(* PLC project Garden Watering, CODESYS CODESYS V3.5 SP14 Patch 1, author Toni Kucic *)
(* stored: creationDateTime 2019-07-15T20:33:55.3489661, version 1.0, modificationDateTime 2019-07-15T20:33:55.2060528, organization TK Automation *)

PROGRAM xc02_GardenWatering
  VAR
    vFlowersXY : ARRAY[0..59, 0..1] OF INT := [276, 253, 381, 253, 486, 253, 591, 253, 696, 253, 801, 253, 906, 253, 1011, 253, 1116, 253, 1221, 253, 276, 354, 381, 354, 486, 354, 591, 354, 696, 354, 801, 354, 906, 354, 1011, 354, 1116, 354, 1221, 354, 276, 455, 381, 455, 486, 455, 591, 455, 696, 455, 801, 455, 906, 455, 1011, 455, 1116, 455, 1221, 455, 276, 556, 381, 556, 486, 556, 591, 556, 696, 556, 801, 556, 906, 556, 1011, 556, 1116, 556, 1221, 556, 276, 667, 381, 667, 486, 667, 591, 667, 696, 667, 801, 667, 906, 667, 1011, 667, 1116, 667, 1221, 667, 276, 768, 381, 768, 486, 768, 591, 768, 696, 768, 801, 768, 906, 768, 1011, 768, 1116, 768, 1221, 768];
    vManual : BOOL;  (* Coordinates of flowers in format Flower0 -x,y *)
    vXCMD : REAL;
    vYCMD : REAL;
    i : INT;
    Watering : TON;
    ActuatorOverFlower : CollisionDetection;
  END_VAR

                    (* Control from the graphics *)
IF NOT xgv02.Remote THEN
	xgv02.HorizontalLeft := xgv02.HMIDownLeft OR xgv02.HMILeft OR xgv02.HMIUpLeft;
	xgv02.HorizontalRight := xgv02.HMIDownRight OR xgv02.HMIRight OR xgv02.HMIUpRight;
	xgv02.VerticalUp := xgv02.HMIUpLeft OR xgv02.HMIUp OR xgv02.HMIUpRight;
	xgv02.VerticalDown := xgv02.HMIDownLeft OR xgv02.HMIDown OR xgv02.HMIDownRight;
	xgv02.OpenWaterValve := xgv02.HMIOpenWater;
END_IF;

(* Coordinate control *)
IF xgv02.Remote AND vManual THEN
	vXCMD := xgv02.HMICoorXCmd;
	vYCMD := xgv02.HMICoorYCmd;
ELSE
	xgv02.HMICoorXCmd := xgv02.PositionX;
	xgv02.HMICoorYCmd := xgv02.PositionY;
END_IF

(* Full automatic algorithm *)
IF xgv02.Remote AND NOT vManual THEN
	vXCMD := vFlowersXY[i,0]+ 30;
	vYCMD := vFlowersXY[i,1]+ 30;
	
	ActuatorOverFlower(
		xcor1:= xgv02.PositionX, 
		ycor1:= xgv02.PositionY, 
		height1:= 10, 
		width1:= 10, 
		xcor2:= vFlowersXY[i,0], 
		ycor2:= vFlowersXY[i,1], 
		height2:= 70, 
		width2:= 70);
		
	IF 	ActuatorOverFlower.isCollision THEN
		Watering(IN:=TRUE, PT:=T#3S);
		xgv02.OpenWaterValve := TRUE;
	END_IF;
	IF ActuatorOverFlower.isCollision AND Watering.Q THEN
		Watering(IN := FALSE);
		xgv02.OpenWaterValve:= FALSE;
		i:= i + 1;	
	END_IF
END_IF
IF i = 59 THEN
	i := 0;
END_IF

(* Actual motor movement section *)
IF xgv02.Remote THEN
	IF vXCMD > xgv02.PositionX - 2 THEN
		xgv02.HorizontalLeft := FALSE;
		xgv02.HorizontalRight := TRUE;
	ELSIF vXCMD < xgv02.PositionX + 2 THEN
		xgv02.HorizontalLeft := TRUE;
		xgv02.HorizontalRight := FALSE;
	ELSE
		xgv02.HorizontalLeft := FALSE;
		xgv02.HorizontalRight := FALSE;
	END_IF;
	
	IF vYCMD < xgv02.PositionY - 2THEN
		xgv02.VerticalUp := TRUE;
		xgv02.VerticalDown := FALSE;
	ELSIF vYCMD > xgv02.PositionY + 2 THEN
		xgv02.VerticalUp := FALSE;
		xgv02.VerticalDown := TRUE;
	ELSE
		xgv02.VerticalUp := FALSE;
		xgv02.VerticalDown := FALSE;
	END_IF;
END_IF;

	

                  
END_PROGRAM

PROGRAM xsim02
  VAR
    CollisionDetector : CollisionDetection;
    FlowerDeathTimer : TON;
    vResetSIM : BOOL;
    vFlowers : ARRAY[0..59] OF DWORD := [60(16#FF73B98B)];
    i : INT;
    vFlowersXY : ARRAY[0..59, 0..1] OF INT := [276, 253, 381, 253, 486, 253, 591, 253, 696, 253, 801, 253, 906, 253, 1011, 253, 1116, 253, 1221, 253, 276, 354, 381, 354, 486, 354, 591, 354, 696, 354, 801, 354, 906, 354, 1011, 354, 1116, 354, 1221, 354, 276, 455, 381, 455, 486, 455, 591, 455, 696, 455, 801, 455, 906, 455, 1011, 455, 1116, 455, 1221, 455, 276, 556, 381, 556, 486, 556, 591, 556, 696, 556, 801, 556, 906, 556, 1011, 556, 1116, 556, 1221, 556, 276, 667, 381, 667, 486, 667, 591, 667, 696, 667, 801, 667, 906, 667, 1011, 667, 1116, 667, 1221, 667, 276, 768, 381, 768, 486, 768, 591, 768, 696, 768, 801, 768, 906, 768, 1011, 768, 1116, 768, 1221, 768];
  END_VAR

                    (* If the plaform covers the flower it will reset its color to initial *)
FOR i:=0 TO 59 BY 1 DO
	CollisionDetector(
		xcor1:= xgv02.PositionX, 
		ycor1:= xgv02.PositionY, 
		height1:= 10, 
		width1:= 10, 
		xcor2:= vFlowersXY[i,0], 
		ycor2:= vFlowersXY[i,1], 
		height2:= 70 , 
		width2:= 70);
	IF CollisionDetector.isCollision AND xgv02.OpenWaterValve THEN
		vFlowers[i] := 16#FF73B98B;
	END_IF
END_FOR

FlowerDeathTimer(IN:=TRUE, PT:=T#60S);
(* Flowers fade its color *)
IF FlowerDeathTimer.Q THEN
	FOR i:=0 TO 59 BY 1 DO
		IF vFlowers[i] > 16#0073B98B THEN
			vFlowers[i] := vFlowers[i] - 16#01000000;
		END_IF;
	END_FOR
	FlowerDeathTimer.IN := FALSE;
END_IF;


                  
END_PROGRAM

FUNCTION_BLOCK Servo
  VAR_INPUT
    CmdFwd : BOOL := FALSE;
    CmdRev : BOOL := FALSE;
    PulseWidth : TIME := TIME#100ms;  (* Width of a pulse from the hall effect sensor when its above magnetic surface *)
  END_VAR
  VAR_OUTPUT
    S1 : BOOL := FALSE;
    S2 : BOOL := FALSE;
  END_VAR
  VAR
    tofS2 : TOF;
    tonS2 : TON;
    blink : BLINK;
    blinkOld : BOOL;
    vStartBlinker : BOOL;
  END_VAR

                    vStartBlinker := (CmdFwd OR CmdRev) AND NOT (CmdFwd AND CmdRev);
Blink(ENABLE := vStartBlinker, TIMELOW:= PulseWidth, TIMEHIGH := PulseWidth);

tonS2(IN := blink.OUT, PT:=PulseWidth/2);
tofS2(IN := NOT tonS2.Q AND blinkOld, PT:=PulseWidth/2);
 
blinkOld := tonS2.Q;

IF CmdFwd THEN
	S1 := blink.OUT;
	S2 := tonS2.Q OR tofS2.Q;
ELSIF CmdRev THEN
	S1 := tonS2.Q OR tofS2.Q;
	S2 := blink.OUT;
END_IF
                  
END_FUNCTION_BLOCK

PROGRAM xc02_GardenWatering_Encoder
  VAR
    HorizontalAxis : Servo;
    VerticalAxis : Servo;
    rtHIncrement : R_TRIG;
    rtHDecrement : R_TRIG;
    rtVIncrement : R_TRIG;
    rtVDecrement : R_TRIG;
    vHorizontalS1Old : BOOL;
    vHorizontalS2Old : BOOL;
    vVerticalS1Old : BOOL;
    vVerticalS2Old : BOOL;
    PositionCounterVerticalAxis : CTUD;
    vHorizontalPos : DINT;
    PositionCounterHorizontalAxis : CTUD;
    vVerticalPos : WORD;
    vPositionX : REAL;
    vPositionY : REAL;
    vHorizontalLimit : BOOL;
    vVerticalLimit : BOOL;
    vPlatformActualPosX : REAL;
    vPlatformActualPosY : REAL;
  END_VAR

                    (* The actual servos that move the watering equipment *)
vHorizontalLimit := (vPositionX >= 940 AND NOT xgv02.HorizontalLeft)
				  OR (vPositionX <= 0 AND NOT xgv02.HorizontalRight);
vVerticalLimit := (vPositionY >= 500 AND NOT xgv02.VerticalUp)
			    OR (vPositionY <= 0 AND NOT xgv02.VerticalDown);

(* Maximum range - 940 steps *)
HorizontalAxis(
	CmdFwd:= xgv02.HorizontalRight AND NOT vHorizontalLimit, 
	CmdRev:= xgv02.HorizontalLeft AND NOT vHorizontalLimit, 
	PulseWidth:= T#0.1S , 
	S1=> xgv02.HorizontalS1, 
	S2=> xgv02.HorizontalS2);
	
(* Maximum range - 500 steps *)	
VerticalAxis(
	CmdFwd:= xgv02.VerticalDown AND NOT vVerticalLimit, 
	CmdRev:= xgv02.VerticalUp AND NOT vVerticalLimit, 
	PulseWidth:= T#0.1S , 
	S1=> xgv02.VerticalS1, 
	S2=> xgv02.VerticalS2);

IF xgv02.HorizontalS1 <> vHorizontalS1Old THEN
	IF xgv02.HorizontalS1 <> xgv02.HorizontalS2 THEN
		rtHIncrement(CLK:=TRUE);
	ELSE
		rtHDecrement(CLK:=TRUE);
	END_IF
ELSE
	rtHIncrement(CLK:=FALSE);
	rtHDecrement(CLK:=FALSE);
END_IF

IF xgv02.VerticalS1 <> vVerticalS1Old THEN
	IF xgv02.VerticalS1 <> xgv02.VerticalS2 THEN
		rtVIncrement(CLK:=TRUE);
	ELSE
		rtVDecrement(CLK:=TRUE);
	END_IF
ELSE
	rtVIncrement(CLK:=FALSE);
	rtVDecrement(CLK:=FALSE);
END_IF

PositionCounterHorizontalAxis(
	CU:= rtHIncrement.Q, 
	CD:= rtHDecrement.Q, 
	CV=> vHorizontalPos);

PositionCounterVerticalAxis(
	CU:= rtVIncrement.Q, 
	CD:= rtVDecrement.Q, 
	CV=> vVerticalPos);
	
(* Position of the system in the graphics*)
(* For every 1 pulses we move 5 px *)
vPositionX := (DINT_TO_REAL(vHorizontalPos)/ 1) * 5;
vPositionY := (DINT_TO_REAL(vVerticalPos)/ 1) * 5;
	
vHorizontalS1Old := xgv02.HorizontalS1;
vVerticalS1Old := xgv02.VerticalS1;
(* This is to counter the starting offset in the graphics *)
vPlatformActualPosX := 307 + vPositionX;
vPlatformActualPosY := 279 + vPositionY;

(* Send the platform position to other programs *)
xgv02.PositionX := vPlatformActualPosX;
xgv02.PositionY := vPlatformActualPosY;
                  
END_PROGRAM

CONFIGURATION SoftPLC
  RESOURCE Application ON PLC
    {attribute 'qualified_only'}
    VAR_GLOBAL  (* xgv02 *)
      HorizontalS1 : BOOL;  (* Configuration Inputs *)
      HorizontalS2 : BOOL;
      VerticalS1 : BOOL;
      VerticalS2 : BOOL;
      PositionX : REAL;  (* Data from encoder *)
      PositionY : REAL;
      HMIUp : BOOL;  (* HMI *)
      HMIDown : BOOL;
      HMIRight : BOOL;
      HMILeft : BOOL;
      HMIUpRight : BOOL;
      HMIUpLeft : BOOL;
      HMIDownRight : BOOL;
      HMIDownLeft : BOOL;
      HMICoorXCmd : REAL;
      HMICoorYCmd : REAL;
      HMIOpenWater : BOOL;
      Remote : BOOL;
      Reset : BOOL;
      HorizontalRight : BOOL;  (* Outputs *)
      HorizontalLeft : BOOL;
      VerticalUp : BOOL;
      VerticalDown : BOOL;
      OpenWaterValve : BOOL;
    END_VAR
    TASK VISU_TASK(INTERVAL := T#50ms, PRIORITY := 31);
    TASK xsim02(INTERVAL := T#20ms, PRIORITY := 2);
    TASK xc02_Task(INTERVAL := T#20ms, PRIORITY := 1);
    PROGRAM VisuElems.Visu_Prg WITH VISU_TASK : VisuElems.Visu_Prg;
    PROGRAM xsim02 WITH xsim02 : xsim02;
    PROGRAM xc02_GardenWatering WITH xc02_Task : xc02_GardenWatering;
    PROGRAM xc02_GardenWatering_Encoder WITH xc02_Task : xc02_GardenWatering_Encoder;
  END_RESOURCE
END_CONFIGURATION
